(* IEC 61131-3 sources: repolevel_ST_code_completion/dataset/generation_context_ground_truth/Robotics_DynamicModel, 15 files *)

(* ---- SMC_Frame_ApplyWrench.st ---- *)
VAR
    mR_ : SM3M.SMC_Matrix3;
    wTmp0 : SM3M.SMC_VECTOR3D;
    wTmp1 : SM3M.SMC_VECTOR3D;
END_VAR

/// Applies a coordinate transformation T_ab to a wrench vector F_a in se(3).
///       |mR^T  mR^T*[vT]^T|
/// F_b = |                 | F_a
///       | 0         mR^T  |
FUNCTION SMC_Frame_ApplyWrench
VAR_IN_OUT
    /// Wrench vector in b frame coordinates.
	F_b : WrenchVec;
END_VAR
VAR_IN_OUT CONSTANT
    /// Orientation and position of the b frame
    /// in a frame coordinates.
	T_ab : SM3M.SMC_Frame;
    /// Wrench vector in a frame coordinates.
	F_a : WrenchVec;
END_VAR
VAR
    mR_ : SM3M.SMC_Matrix3;
    wTmp0 : SM3M.SMC_VECTOR3D;
    wTmp1 : SM3M.SMC_VECTOR3D;
END_VAR

(* ---- DynModel_Scara2_Z.st ---- *)
VAR CONSTANT
	/// Degrees of freedom.
	DOF : DINT := 3;
	/// All length values in [m]
	armOneLength : LREAL := 0.4;
	armTwoLength : LREAL := 0.3;
	baseHeight : LREAL := 0.6;
	armOneHeight : LREAL := 0.06;
	armTwoHeight : LREAL := 0.06;
	zAxisLength : LREAL := 0.3;
	zAxisOffset : LREAL := -0.05;
	/// All mass values in [kg]
	armOneMass : LREAL := 3;
	armTwoMass : LREAL := 4;
	zAxisMass : LREAL := 1;

	/// The home position of all link frames. |aM[i]| contains
    /// the frame of the ith link expressed in the coordinates of the
    /// (i-1)th link frame.
    /// All frames are expected to be situated at the link's center
    /// of mass.
    m_aM : ARRAY[0..SMRB.MAX_VEC_DIM] OF SM3M.SMC_Frame := [
        /// All values of vT in [m]
        ///
        /// The center of mass of arm 1 expressed in the base coordinate system 0:
        (mR:= (
            aElems:= [
                1, 0, 0,
                0, -1, 0,
                0, 0, -1]),
         vT:= (dX:= armOneLength / 2.0, dY:= 0, dZ:= baseHeight + armOneHeight / 2.0)),
        /// The center of mass of arm 2 expressed in the coordinate system of arm 1:
        (mR:= (
            aElems:= [
                1, 0, 0,
                0, 1, 0,
                0, 0, 1]),
         vT:= (dX:= armOneLength / 2.0 + armTwoLength / 2.0, dY:= 0, dZ:= armOneHeight / 2.0 + armTwoHeight / 2.0)),
        /// The center of mass of the z-axis expressed in the coordinate system of arm 2:
        (mR:= (
            aElems:= [
                1, 0, 0,
                0, 1, 0,
                0, 0, 1]),
         vT:= (dX:= armTwoLength / 2.0, dY:= 0, dZ:= zAxisLength / 2.0 - armTwoHeight / 2.0 + zAxisOffset)),
        /// One additional array entry, to handle an arbitrary load at the TCP, expressed
		/// in the coordinate system of the z-axis.
        (mR:= (
            aElems:= [
                1, 0, 0,
                0, 1, 0,
                0, 0, 1]),
         vT:= (dX:= 0, dY:= 0, dZ:= - zAxisLength / 2.0))];

	/// The spatial inertia matrices of all links, expressed in the
    /// respectives link's frame.
    m_aG : ARRAY[0..SMRB.MAX_VEC_DIM-1] OF SMDYN.DynSpatialInertia := [
        /// All inertia values in [kg m²]
        /// and all mass values in [kg]
        /// Arm 1
        (I:= (
            aElems:= [
                0, 0, 0,
                0, 1/12.0 * armOneMass * armOneLength * armOneLength, 0,
                0, 0, 1/12.0 * armOneMass * armOneLength * armOneLength]),
         m:= armOneMass),
        /// Arm 2
        (I:= (
            aElems:= [
                0, 0, 0,
                0, 1/12.0 * armTwoMass * armTwoLength * armTwoLength, 0,
                0, 0, 1/12.0 * armTwoMass * armTwoLength * armTwoLength]),
         m:= armTwoMass),
        /// z-axis
        (I:= (
            aElems:= [
                1/12.0 * zAxisMass * zAxisLength * zAxisLength, 0, 0,
                0, 1/12.0 * zAxisMass * zAxisLength * zAxisLength, 0,
                0, 0, 0]),
         m:= zAxisMass)];

	/// The screw axes of all joints, expressed in the base frame.
    m_aS : ARRAY[0..SMRB.MAX_VEC_DIM-1] OF TwistVec := [
		/// Angular velocities in [rad/s] and linear velocities in [m/s].
        /// Screw axis of arm 1
        (w:= (dX:= 0, dY:= 0, dZ:= 1),
         v:= (dX:= 0, dY:= 0, dZ:= 0)),
        /// Screw axis of arm 2
        (w:= (dX:= 0, dY:= 0, dZ:= 1),
         v:= (dX:= 0, dY:= -armOneLength, dZ:= 0)),
        /// Screw axis of the z-axis
        (w:= (dX:= 0, dY:= 0, dZ:= 0),
         v:= (dX:= 0, dY:= 0, dZ:= 1))];
END_VAR
VAR
    /// The home position of all link frames. |m_aM_inv[i]| contains
    /// the frame of the (i-1) link expressed in the coordinates of the
    /// ith link frame.
    /// All frames are expected to be situated at the link's center
    /// of mass.
    m_aM_inv : ARRAY[0..SM3M.SMC_MAX_VEC_DIM] OF SM3M.SMC_Frame;
    /// The screw axes of all joints, expressed in the link's frame.
    m_aA : ARRAY[0..SM3M.SMC_MAX_VEC_DIM-1] OF TwistVec;
END_VAR

(* ---- DynModel_Scara2_Z_AxesStateToTorque.st ---- *)
VAR
	m_aM_inv : ARRAY[0..SM3M.SMC_MAX_VEC_DIM] OF SM3M.SMC_Frame;
    /// The screw axes of all joints, expressed in the link's frame.
    m_aA : ARRAY[0..SM3M.SMC_MAX_VEC_DIM-1] OF TwistVec;
    convertedAxesState : SM3M.SMC_DynVecState;
	i : DINT;
END_VAR

VAR CONSTANT
/// Degrees of freedom.
	DOF : DINT := 3;
	/// All length values in [m]
	armOneLength : LREAL := 0.4;
	armTwoLength : LREAL := 0.3;
	baseHeight : LREAL := 0.6;
	armOneHeight : LREAL := 0.06;
	armTwoHeight : LREAL := 0.06;
	zAxisLength : LREAL := 0.3;
	zAxisOffset : LREAL := -0.05;
	/// All mass values in [kg]
	armOneMass : LREAL := 3;
	armTwoMass : LREAL := 4;
	zAxisMass : LREAL := 1;

	/// The home position of all link frames. |aM[i]| contains
    /// the frame of the ith link expressed in the coordinates of the
    /// (i-1)th link frame.
    /// All frames are expected to be situated at the link's center
    /// of mass.
    m_aM : ARRAY[0..SMRB.MAX_VEC_DIM] OF SM3M.SMC_Frame := [
        /// All values of vT in [m]
        ///
        /// The center of mass of arm 1 expressed in the base coordinate system 0:
        (mR:= (
            aElems:= [
                1, 0, 0,
                0, -1, 0,
                0, 0, -1]),
         vT:= (dX:= armOneLength / 2.0, dY:= 0, dZ:= baseHeight + armOneHeight / 2.0)),
        /// The center of mass of arm 2 expressed in the coordinate system of arm 1:
        (mR:= (
            aElems:= [
                1, 0, 0,
                0, 1, 0,
                0, 0, 1]),
         vT:= (dX:= armOneLength / 2.0 + armTwoLength / 2.0, dY:= 0, dZ:= armOneHeight / 2.0 + armTwoHeight / 2.0)),
        /// The center of mass of the z-axis expressed in the coordinate system of arm 2:
        (mR:= (
            aElems:= [
                1, 0, 0,
                0, 1, 0,
                0, 0, 1]),
         vT:= (dX:= armTwoLength / 2.0, dY:= 0, dZ:= zAxisLength / 2.0 - armTwoHeight / 2.0 + zAxisOffset)),
        /// One additional array entry, to handle an arbitrary load at the TCP, expressed
		/// in the coordinate system of the z-axis.
        (mR:= (
            aElems:= [
                1, 0, 0,
                0, 1, 0,
                0, 0, 1]),
         vT:= (dX:= 0, dY:= 0, dZ:= - zAxisLength / 2.0))];

	/// The spatial inertia matrices of all links, expressed in the
    /// respectives link's frame.
    m_aG : ARRAY[0..SMRB.MAX_VEC_DIM-1] OF SMDYN.DynSpatialInertia := [
        /// All inertia values in [kg m²]
        /// and all mass values in [kg]
        /// Arm 1
        (I:= (
            aElems:= [
                0, 0, 0,
                0, 1/12.0 * armOneMass * armOneLength * armOneLength, 0,
                0, 0, 1/12.0 * armOneMass * armOneLength * armOneLength]),
         m:= armOneMass),
        /// Arm 2
        (I:= (
            aElems:= [
                0, 0, 0,
                0, 1/12.0 * armTwoMass * armTwoLength * armTwoLength, 0,
                0, 0, 1/12.0 * armTwoMass * armTwoLength * armTwoLength]),
         m:= armTwoMass),
        /// z-axis
        (I:= (
            aElems:= [
                1/12.0 * zAxisMass * zAxisLength * zAxisLength, 0, 0,
                0, 1/12.0 * zAxisMass * zAxisLength * zAxisLength, 0,
                0, 0, 0]),
         m:= zAxisMass)];

	/// The screw axes of all joints, expressed in the base frame.
    m_aS : ARRAY[0..SMRB.MAX_VEC_DIM-1] OF TwistVec := [
		/// Angular velocities in [rad/s] and linear velocities in [m/s].
        /// Screw axis of arm 1
        (w:= (dX:= 0, dY:= 0, dZ:= 1),
         v:= (dX:= 0, dY:= 0, dZ:= 0)),
        /// Screw axis of arm 2
        (w:= (dX:= 0, dY:= 0, dZ:= 1),
         v:= (dX:= 0, dY:= -armOneLength, dZ:= 0)),
        /// Screw axis of the z-axis
        (w:= (dX:= 0, dY:= 0, dZ:= 0),
         v:= (dX:= 0, dY:= 0, dZ:= 1))];
END_VAR

ConvertAxesState(convertedAxesState, axesState);

SolveOpenChainDynamics(
	torque:= torque,
	uv:= convertedAxesState,
	g:= addParams.g,
	load:= addParams.load);

AxesStateToTorque := SMC_NO_ERROR;

(* ---- DynModel_Scara2_Z_ConvertAxesState.st ---- *)
VAR
    i : DINT;
	m_aM_inv : ARRAY[0..SM3M.SMC_MAX_VEC_DIM] OF SM3M.SMC_Frame;
    /// The screw axes of all joints, expressed in the link's frame.
    m_aA : ARRAY[0..SM3M.SMC_MAX_VEC_DIM-1] OF TwistVec;
END_VAR
VAR CONSTANT
/// Degrees of freedom.
	DOF : DINT := 3;
	/// All length values in [m]
	armOneLength : LREAL := 0.4;
	armTwoLength : LREAL := 0.3;
	baseHeight : LREAL := 0.6;
	armOneHeight : LREAL := 0.06;
	armTwoHeight : LREAL := 0.06;
	zAxisLength : LREAL := 0.3;
	zAxisOffset : LREAL := -0.05;
	/// All mass values in [kg]
	armOneMass : LREAL := 3;
	armTwoMass : LREAL := 4;
	zAxisMass : LREAL := 1;

	/// The home position of all link frames. |aM[i]| contains
    /// the frame of the ith link expressed in the coordinates of the
    /// (i-1)th link frame.
    /// All frames are expected to be situated at the link's center
    /// of mass.
    m_aM : ARRAY[0..SMRB.MAX_VEC_DIM] OF SM3M.SMC_Frame := [
        /// All values of vT in [m]
        ///
        /// The center of mass of arm 1 expressed in the base coordinate system 0:
        (mR:= (
            aElems:= [
                1, 0, 0,
                0, -1, 0,
                0, 0, -1]),
         vT:= (dX:= armOneLength / 2.0, dY:= 0, dZ:= baseHeight + armOneHeight / 2.0)),
        /// The center of mass of arm 2 expressed in the coordinate system of arm 1:
        (mR:= (
            aElems:= [
                1, 0, 0,
                0, 1, 0,
                0, 0, 1]),
         vT:= (dX:= armOneLength / 2.0 + armTwoLength / 2.0, dY:= 0, dZ:= armOneHeight / 2.0 + armTwoHeight / 2.0)),
        /// The center of mass of the z-axis expressed in the coordinate system of arm 2:
        (mR:= (
            aElems:= [
                1, 0, 0,
                0, 1, 0,
                0, 0, 1]),
         vT:= (dX:= armTwoLength / 2.0, dY:= 0, dZ:= zAxisLength / 2.0 - armTwoHeight / 2.0 + zAxisOffset)),
        /// One additional array entry, to handle an arbitrary load at the TCP, expressed
		/// in the coordinate system of the z-axis.
        (mR:= (
            aElems:= [
                1, 0, 0,
                0, 1, 0,
                0, 0, 1]),
         vT:= (dX:= 0, dY:= 0, dZ:= - zAxisLength / 2.0))];

	/// The spatial inertia matrices of all links, expressed in the
    /// respectives link's frame.
    m_aG : ARRAY[0..SMRB.MAX_VEC_DIM-1] OF SMDYN.DynSpatialInertia := [
        /// All inertia values in [kg m²]
        /// and all mass values in [kg]
        /// Arm 1
        (I:= (
            aElems:= [
                0, 0, 0,
                0, 1/12.0 * armOneMass * armOneLength * armOneLength, 0,
                0, 0, 1/12.0 * armOneMass * armOneLength * armOneLength]),
         m:= armOneMass),
        /// Arm 2
        (I:= (
            aElems:= [
                0, 0, 0,
                0, 1/12.0 * armTwoMass * armTwoLength * armTwoLength, 0,
                0, 0, 1/12.0 * armTwoMass * armTwoLength * armTwoLength]),
         m:= armTwoMass),
        /// z-axis
        (I:= (
            aElems:= [
                1/12.0 * zAxisMass * zAxisLength * zAxisLength, 0, 0,
                0, 1/12.0 * zAxisMass * zAxisLength * zAxisLength, 0,
                0, 0, 0]),
         m:= zAxisMass)];

	/// The screw axes of all joints, expressed in the base frame.
    m_aS : ARRAY[0..SMRB.MAX_VEC_DIM-1] OF TwistVec := [
		/// Angular velocities in [rad/s] and linear velocities in [m/s].
        /// Screw axis of arm 1
        (w:= (dX:= 0, dY:= 0, dZ:= 1),
         v:= (dX:= 0, dY:= 0, dZ:= 0)),
        /// Screw axis of arm 2
        (w:= (dX:= 0, dY:= 0, dZ:= 1),
         v:= (dX:= 0, dY:= -armOneLength, dZ:= 0)),
        /// Screw axis of the z-axis
        (w:= (dX:= 0, dY:= 0, dZ:= 0),
         v:= (dX:= 0, dY:= 0, dZ:= 1))];
END_VAR

FOR i := 0 TO 2 DO
	CASE i OF
		0, 1:
			convertedAxesState.v.a[i] := axesState.v.a[i] * SM3M.SMC_FACTOR_DEG_TO_RAD;
			convertedAxesState.v_s.a[i] := axesState.v_s.a[i] * SM3M.SMC_FACTOR_DEG_TO_RAD;
			convertedAxesState.v_ss.a[i] := axesState.v_ss.a[i] * SM3M.SMC_FACTOR_DEG_TO_RAD;

		2:
			convertedAxesState.v.a[i] := axesState.v.a[i];
			convertedAxesState.v_s.a[i] := axesState.v_s.a[i];
			convertedAxesState.v_ss.a[i] := axesState.v_ss.a[i];
	END_CASE
END_FOR

convertedAxesState.v.n :=
convertedAxesState.v_s.n :=
convertedAxesState.v_ss.n := 3;

(* ---- DynModel_Scara2_Z_Init.st ---- *)
VAR CONSTANT
/// Degrees of freedom.
	DOF : DINT := 3;
	/// All length values in [m]
	armOneLength : LREAL := 0.4;
	armTwoLength : LREAL := 0.3;
	baseHeight : LREAL := 0.6;
	armOneHeight : LREAL := 0.06;
	armTwoHeight : LREAL := 0.06;
	zAxisLength : LREAL := 0.3;
	zAxisOffset : LREAL := -0.05;
	/// All mass values in [kg]
	armOneMass : LREAL := 3;
	armTwoMass : LREAL := 4;
	zAxisMass : LREAL := 1;

	/// The home position of all link frames. |aM[i]| contains
    /// the frame of the ith link expressed in the coordinates of the
    /// (i-1)th link frame.
    /// All frames are expected to be situated at the link's center
    /// of mass.
    m_aM : ARRAY[0..SMRB.MAX_VEC_DIM] OF SM3M.SMC_Frame := [
        /// All values of vT in [m]
        ///
        /// The center of mass of arm 1 expressed in the base coordinate system 0:
        (mR:= (
            aElems:= [
                1, 0, 0,
                0, -1, 0,
                0, 0, -1]),
         vT:= (dX:= armOneLength / 2.0, dY:= 0, dZ:= baseHeight + armOneHeight / 2.0)),
        /// The center of mass of arm 2 expressed in the coordinate system of arm 1:
        (mR:= (
            aElems:= [
                1, 0, 0,
                0, 1, 0,
                0, 0, 1]),
         vT:= (dX:= armOneLength / 2.0 + armTwoLength / 2.0, dY:= 0, dZ:= armOneHeight / 2.0 + armTwoHeight / 2.0)),
        /// The center of mass of the z-axis expressed in the coordinate system of arm 2:
        (mR:= (
            aElems:= [
                1, 0, 0,
                0, 1, 0,
                0, 0, 1]),
         vT:= (dX:= armTwoLength / 2.0, dY:= 0, dZ:= zAxisLength / 2.0 - armTwoHeight / 2.0 + zAxisOffset)),
        /// One additional array entry, to handle an arbitrary load at the TCP, expressed
		/// in the coordinate system of the z-axis.
        (mR:= (
            aElems:= [
                1, 0, 0,
                0, 1, 0,
                0, 0, 1]),
         vT:= (dX:= 0, dY:= 0, dZ:= - zAxisLength / 2.0))];

	/// The spatial inertia matrices of all links, expressed in the
    /// respectives link's frame.
    m_aG : ARRAY[0..SMRB.MAX_VEC_DIM-1] OF SMDYN.DynSpatialInertia := [
        /// All inertia values in [kg m²]
        /// and all mass values in [kg]
        /// Arm 1
        (I:= (
            aElems:= [
                0, 0, 0,
                0, 1/12.0 * armOneMass * armOneLength * armOneLength, 0,
                0, 0, 1/12.0 * armOneMass * armOneLength * armOneLength]),
         m:= armOneMass),
        /// Arm 2
        (I:= (
            aElems:= [
                0, 0, 0,
                0, 1/12.0 * armTwoMass * armTwoLength * armTwoLength, 0,
                0, 0, 1/12.0 * armTwoMass * armTwoLength * armTwoLength]),
         m:= armTwoMass),
        /// z-axis
        (I:= (
            aElems:= [
                1/12.0 * zAxisMass * zAxisLength * zAxisLength, 0, 0,
                0, 1/12.0 * zAxisMass * zAxisLength * zAxisLength, 0,
                0, 0, 0]),
         m:= zAxisMass)];

	/// The screw axes of all joints, expressed in the base frame.
    m_aS : ARRAY[0..SMRB.MAX_VEC_DIM-1] OF TwistVec := [
		/// Angular velocities in [rad/s] and linear velocities in [m/s].
        /// Screw axis of arm 1
        (w:= (dX:= 0, dY:= 0, dZ:= 1),
         v:= (dX:= 0, dY:= 0, dZ:= 0)),
        /// Screw axis of arm 2
        (w:= (dX:= 0, dY:= 0, dZ:= 1),
         v:= (dX:= 0, dY:= -armOneLength, dZ:= 0)),
        /// Screw axis of the z-axis
        (w:= (dX:= 0, dY:= 0, dZ:= 0),
         v:= (dX:= 0, dY:= 0, dZ:= 1))];
END_VAR
VAR
    i : DINT;
    M_ib_ : SM3M.SMC_Frame;
    M_ib : SM3M.SMC_Frame; // base frame expressed in ith frame
    m_aM_inv : ARRAY[0..SM3M.SMC_MAX_VEC_DIM] OF SM3M.SMC_Frame;
    /// The screw axes of all joints, expressed in the link's frame.
    m_aA : ARRAY[0..SM3M.SMC_MAX_VEC_DIM-1] OF TwistVec;
END_VAR

/// Initialize constant parameters that are used by the open chain dynamics algorithm:
/// - Calculate the inverse frames of the center of mass positions m_aM_inv from the
/// given center of mass positions m_aM.
/// - Calculate the screw axes of all joints m_aA (expressed in the link´s frame)
/// from the given screw axes m_aS, which are expressed in the base frame.
M_ib := SM3M.SMC_Math_Global_Constants.SMC_FRAME_IDENTITY;
i := 0;
WHILE i < DOF DO
    SM3M.SMC_Frame_Inverse(m_aM_inv[i], m_aM[i]);

    SM3M.SMC_Frame_Mult(M_ib_, m_aM_inv[i], M_ib);
    M_ib := M_ib_;
    SMC_Frame_ApplyTwist(m_aA[i], M_ib, m_aS[i]);

    i := i + 1;
END_WHILE

SM3M.SMC_Frame_Inverse(m_aM_inv[DOF], m_aM[DOF]);

(* ---- DynModel_Scara2_Z_SolveOpenChainDynamics.st ---- *)
VAR
    T : ARRAY[0..SM3M.SMC_MAX_VEC_DIM] OF SM3M.SMC_Frame;
    V : ARRAY[0..SM3M.SMC_MAX_VEC_DIM] OF TwistVec;
    V_t : ARRAY[0..SM3M.SMC_MAX_VEC_DIM] OF TwistVec;
    F : ARRAY[0..SM3M.SMC_MAX_VEC_DIM] OF WrenchVec;

    T_uq : SM3M.SMC_Frame;
    V_uq_s : TwistVec;
    V_t_uq_ss : TwistVec;
    V_prev : TwistVec;
    V_t_prev : TwistVec;
    V_t_brack : TwistVec;
    F_prev : WrenchVec;
    F_V : WrenchVec;
    F_V_t : WrenchVec;
    F_brack : WrenchVec;
    i : DINT;

    T_load_inv_Flange : SM3M.SMC_Frame;
    T_load_inv : SM3M.SMC_Frame;
    V_load : TwistVec;
    V_t_load : TwistVec;
    F_load : WrenchVec;
    F_V_load : WrenchVec;
    F_V_t_load : WrenchVec;
    F_brack_load : WrenchVec;
    m_aM_inv : ARRAY[0..SM3M.SMC_MAX_VEC_DIM] OF SM3M.SMC_Frame;
    /// The screw axes of all joints, expressed in the link's frame.
    m_aA : ARRAY[0..SM3M.SMC_MAX_VEC_DIM-1] OF TwistVec;
END_VAR
VAR CONSTANT
/// Degrees of freedom.
	DOF : DINT := 3;
	/// All length values in [m]
	armOneLength : LREAL := 0.4;
	armTwoLength : LREAL := 0.3;
	baseHeight : LREAL := 0.6;
	armOneHeight : LREAL := 0.06;
	armTwoHeight : LREAL := 0.06;
	zAxisLength : LREAL := 0.3;
	zAxisOffset : LREAL := -0.05;
	/// All mass values in [kg]
	armOneMass : LREAL := 3;
	armTwoMass : LREAL := 4;
	zAxisMass : LREAL := 1;

	/// The home position of all link frames. |aM[i]| contains
    /// the frame of the ith link expressed in the coordinates of the
    /// (i-1)th link frame.
    /// All frames are expected to be situated at the link's center
    /// of mass.
    m_aM : ARRAY[0..SMRB.MAX_VEC_DIM] OF SM3M.SMC_Frame := [
        /// All values of vT in [m]
        ///
        /// The center of mass of arm 1 expressed in the base coordinate system 0:
        (mR:= (
            aElems:= [
                1, 0, 0,
                0, -1, 0,
                0, 0, -1]),
         vT:= (dX:= armOneLength / 2.0, dY:= 0, dZ:= baseHeight + armOneHeight / 2.0)),
        /// The center of mass of arm 2 expressed in the coordinate system of arm 1:
        (mR:= (
            aElems:= [
                1, 0, 0,
                0, 1, 0,
                0, 0, 1]),
         vT:= (dX:= armOneLength / 2.0 + armTwoLength / 2.0, dY:= 0, dZ:= armOneHeight / 2.0 + armTwoHeight / 2.0)),
        /// The center of mass of the z-axis expressed in the coordinate system of arm 2:
        (mR:= (
            aElems:= [
                1, 0, 0,
                0, 1, 0,
                0, 0, 1]),
         vT:= (dX:= armTwoLength / 2.0, dY:= 0, dZ:= zAxisLength / 2.0 - armTwoHeight / 2.0 + zAxisOffset)),
        /// One additional array entry, to handle an arbitrary load at the TCP, expressed
		/// in the coordinate system of the z-axis.
        (mR:= (
            aElems:= [
                1, 0, 0,
                0, 1, 0,
                0, 0, 1]),
         vT:= (dX:= 0, dY:= 0, dZ:= - zAxisLength / 2.0))];

	/// The spatial inertia matrices of all links, expressed in the
    /// respectives link's frame.
    m_aG : ARRAY[0..SMRB.MAX_VEC_DIM-1] OF SMDYN.DynSpatialInertia := [
        /// All inertia values in [kg m²]
        /// and all mass values in [kg]
        /// Arm 1
        (I:= (
            aElems:= [
                0, 0, 0,
                0, 1/12.0 * armOneMass * armOneLength * armOneLength, 0,
                0, 0, 1/12.0 * armOneMass * armOneLength * armOneLength]),
         m:= armOneMass),
        /// Arm 2
        (I:= (
            aElems:= [
                0, 0, 0,
                0, 1/12.0 * armTwoMass * armTwoLength * armTwoLength, 0,
                0, 0, 1/12.0 * armTwoMass * armTwoLength * armTwoLength]),
         m:= armTwoMass),
        /// z-axis
        (I:= (
            aElems:= [
                1/12.0 * zAxisMass * zAxisLength * zAxisLength, 0, 0,
                0, 1/12.0 * zAxisMass * zAxisLength * zAxisLength, 0,
                0, 0, 0]),
         m:= zAxisMass)];

	/// The screw axes of all joints, expressed in the base frame.
    m_aS : ARRAY[0..SMRB.MAX_VEC_DIM-1] OF TwistVec := [
		/// Angular velocities in [rad/s] and linear velocities in [m/s].
        /// Screw axis of arm 1
        (w:= (dX:= 0, dY:= 0, dZ:= 1),
         v:= (dX:= 0, dY:= 0, dZ:= 0)),
        /// Screw axis of arm 2
        (w:= (dX:= 0, dY:= 0, dZ:= 1),
         v:= (dX:= 0, dY:= -armOneLength, dZ:= 0)),
        /// Screw axis of the z-axis
        (w:= (dX:= 0, dY:= 0, dZ:= 0),
         v:= (dX:= 0, dY:= 0, dZ:= 1))];
END_VAR

SM3M.SMC_V3_Mult(V_t[0].v, g, -1);

T[DOF] := m_aM_inv[DOF];

i := 0;
WHILE i < DOF DO
    SMC_Frame_FromScrewAxisAngle(T_uq, m_aA[i], -uv.v.a[i]);
    SM3M.SMC_Frame_Mult(T[i], T_uq, m_aM_inv[i]);

    SMC_Frame_ApplyTwist(V_prev, T[i], V[i]);
    TwistVec_Scale(V_uq_s, m_aA[i], uv.v_s.a[i]);
    TwistVec_Add(V[i+1], V_prev, V_uq_s);

    SMC_Frame_ApplyTwist(V_t_prev, T[i], V_t[i]);
    Twist_Bracket_Twist(V_t_brack, V[i+1], m_aA[i]);
    TwistVec_Scale(V_t_brack, V_t_brack, uv.v_s.a[i]);
    TwistVec_Scale(V_t_uq_ss, m_aA[i], uv.v_ss.a[i]);
    TwistVec_Add(V_t[i+1], V_t_prev, V_t_brack);
    TwistVec_Add(V_t[i+1], V_t[i+1], V_t_uq_ss);

    i := i + 1;
END_WHILE

SM3M.SMC_Frame_Inverse(T_load_inv_Flange, load.CenterOfMassFrame);
SM3M.SMC_Frame_Mult(T_load_inv, T_load_inv_Flange, T[i]);

SMC_Frame_ApplyTwist(V_load, T_load_inv, V[i]);
SMC_Frame_ApplyTwist(V_t_load, T_load_inv, V_t[i]);
MatSI_ApplyTwist(F_V_t_load, load.Inertia, V_t_load);
MatSI_ApplyTwist(F_V_load, load.Inertia, V_load);
Twist_Bracket_Wrench(F_brack_load, V_load, F_V_load);

WrenchVec_Sub(F_load, F_V_t_load, F_brack_load);
SMC_Frame_ApplyWrench(F[DOF], T_load_inv_Flange, F_load);

WHILE i > 0 DO
    SMC_Frame_ApplyWrench(F_prev, T[i], F[i]);
    MatSI_ApplyTwist(F_V_t, m_aG[i-1], V_t[i]);
    MatSI_ApplyTwist(F_V, m_aG[i-1], V[i]);
    Twist_Bracket_Wrench(F_brack, V[i], F_V);

    WrenchVec_Add(F[i-1], F_prev, F_V_t);
    WrenchVec_Sub(F[i-1], F[i-1], F_brack);

    torque.a[i-1] := Wrench_Dot_Twist(F[i-1], m_aA[i-1]);

    i := i - 1;
END_WHILE

torque.n := DOF;

(* ---- SMC_Frame_ApplyTwist.st ---- *)
VAR
    vTmp : SM3M.SMC_VECTOR3D;
END_VAR

SM3M.SMC_Matrix3_Apply(V_a.w, T_ab.mR, V_b.w);
SM3M.SMC_Matrix3_Apply(V_a.v, T_ab.mR, V_b.v);
SM3M.SMC_V3_Cross(vTmp, T_ab.vT, V_a.w);
SM3M.SMC_V3_Add(V_a.v, V_a.v, vTmp);

(* ---- SMC_Frame_FromScrewAxisAngle.st ---- *)
VAR
    wv : SM3M.SMC_VECTOR3D;
    w2v : SM3M.SMC_VECTOR3D;
    wt : SM3M.SMC_VECTOR3D;
END_VAR

SM3M.SMC_V3_Cross(wv, A.w, A.v);
SM3M.SMC_V3_Cross(w2v, A.w, wv);

SM3M.SMC_V3_Mult(f.vT, A.v, theta);
SM3M.SMC_V3_MAdd(f.vT, f.vT, wv, (1 - COS(theta)));
SM3M.SMC_V3_MAdd(f.vT, f.vT, w2v, (theta - SIN(theta)));

SM3M.SMC_V3_Mult(wt, A.w, theta);
SM3M.SMC_Matrix3_FromAxisAngle(f.mR, wt);

(* ---- SMC_OpenChainKinematics_SolveForward.st ---- *)
VAR
    i : UDINT;
    fTmp : SM3M.SMC_Frame;
    afCur : ARRAY[0..1] OF SM3M.SMC_Frame;
END_VAR

i := TO_UDINT(vJoints.n);
afCur[i AND 1] := fTCP_init;
WHILE i > 0 DO
    SMC_Frame_FromScrewAxisAngle(fTmp, aS[i-1], vJoints.a[i-1]);
    SM3M.SMC_Frame_Mult(afCur[(i-1) AND 1], fTmp, afCur[i AND 1]);

    i := i - 1;
END_WHILE

fTCP := afCur[0];

(* ---- Test_DynModel_Scara2_Z.st ---- *)
VAR
	m_dynModel : DynModel_Scara2_Z;
END_VAR
VAR CONSTANT
	/// Frame of the initial robot position.
	ZERO_TCP_FRAME : SM3M.SMC_Frame := (
        mR:= (
            aElems:= [
                1, 0, 0,
                0, 1, 0,
                0, 0, 1]),
        vT:= (
			dX:= m_dynModel.armOneLength + m_dynModel.armTwoLength,
			dY:= 0,
			dZ:= - m_dynModel.baseHeight - m_dynModel.armOneHeight - m_dynModel.zAxisOffset));
END_VAR

(* ---- Test_DynModel_Scara2_Z_CheckScrewAxis.st ---- *)
VAR
	state : INT;
	done : BOOL;
	error : BOOL;

	axisPos : TRAFO.AXISPOS_REF;
END_VAR
VAR CONSTANT
	EPS : LREAL := 1E-10;
END_VAR

m_dynModel.Init();

WHILE NOT done AND NOT error DO
	CASE state OF
		0:
			axisPos.a0 := 0;	/// [°]
			axisPos.a1 := 0;	/// [°]
			axisPos.a2 := 0;	/// [m]

			IF IsScrewAxisAndKinematicEqual(axisPos, EPS) THEN
				state := state + 10;
			ELSE
				error := TRUE;
			END_IF

		10:
			axisPos.a0 := 0;	/// [°]
			axisPos.a1 := 90;	/// [°]
			axisPos.a2 := 0.03;	/// [m]

			IF IsScrewAxisAndKinematicEqual(axisPos, EPS) THEN
				state := state + 10;
			ELSE
				error := TRUE;
			END_IF

		20:
			axisPos.a0 := 45;	/// [°]
			axisPos.a1 := -50;	/// [°]
			axisPos.a2 := -0.01;/// [m]

			IF IsScrewAxisAndKinematicEqual(axisPos, EPS) THEN
				state := state + 10;
			ELSE
				error := TRUE;
			END_IF

		30:
			done := TRUE;
	END_CASE
END_WHILE

CheckScrewAxis := done AND NOT error;

(* ---- Test_DynModel_Scara2_Z_CheckStandstillTorque.st ---- *)
VAR
	expectedTorque : SM3M.SMC_Vec;
	calculatedTorque : SM3M.SMC_Vec;
	axesState : SM3M.SMC_DynVecState;
	addParams : SMDYN.DynamicsParams;
	i : DINT;
END_VAR
VAR CONSTANT
	EPSILON : LREAL := 1E-10;
END_VAR

m_dynModel.Init();

/// All axes in zero position.
axesState.v.a[0] := 0;
axesState.v.a[1] := 0;
axesState.v.a[2] := 0;
axesState.v.n := axesState.v_s.n := axesState.v_ss.n := 3;

/// Gravitational acceleration in [m/s²]
addParams.g.dZ := 9.81;

/// Expected torque of the revolute axis of arm 1 in [Nm]
expectedTorque.a[0] := 0;
/// Expected torque of the revolute axis of arm 2 in [Nm]
expectedTorque.a[1] := 0;
/// Expected force of the prismatic z-axis in [N]
expectedTorque.a[2] := - m_dynModel.zAxisMass * 9.81;
expectedTorque.n := 3;

m_dynModel.AxesStateToTorque(
	torque:= calculatedTorque,
	axesState:= axesState,
	addParams:= addParams);

CheckStandstillTorque := calculatedTorque.n = expectedTorque.n;
FOR i := 0 TO calculatedTorque.n - 1 DO
	CheckStandstillTorque := CheckStandstillTorque
							 AND_THEN ABS(calculatedTorque.a[i] - expectedTorque.a[i]) <= EPSILON;
END_FOR

(* ---- Test_DynModel_Scara2_Z_IsScrewAxisAndKinematicEqual.st ---- *)
VAR
	getKinematic : MC_ReadKinTransform;
	screwAxisResult : SM3M.SMC_Frame;
	convertedAxisPos : SM3M.SMC_Vec;
	kinematicResult : SM3M.SMC_Frame;
	cdNotUsed : TRAFO.CONFIGDATA;
END_VAR

convertedAxisPos.a[0] := axisPos.a0 * SM3M.SMC_FACTOR_DEG_TO_RAD;
convertedAxisPos.a[1] := axisPos.a1 * SM3M.SMC_FACTOR_DEG_TO_RAD;
convertedAxisPos.a[2] := axisPos.a2;
convertedAxisPos.n := 3;

SMC_OpenChainKinematics_SolveForward(
	fTCP:= screwAxisResult,
	aS:= m_dynModel.m_aS,
	vJoints:= convertedAxisPos,
	fTCP_init:= ZERO_TCP_FRAME);

getKinematic(
	AxisGroup:= AxisGroup,
	Enable:= TRUE);

IF getKinematic.Valid AND_THEN getKinematic.KinTransform <> 0 THEN
	getKinematic.KinTransform.AxesToCartesian(
		f:= kinematicResult,
		cd:= cdNotUsed,
		a:= axisPos);

	IsScrewAxisAndKinematicEqual :=
		ABS(screwAxisResult.vT.dX - kinematicResult.vT.dX) <= epsilon
		AND_THEN ABS(screwAxisResult.vT.dY- kinematicResult.vT.dY) <= epsilon
		AND_THEN ABS(screwAxisResult.vT.dZ - kinematicResult.vT.dZ) <= epsilon;
ELSE
	IsScrewAxisAndKinematicEqual := FALSE;
END_IF

(* ---- Twist_Bracket_Twist.st ---- *)
VAR
    v0 : SM3M.SMC_VECTOR3D;
    v1 : SM3M.SMC_VECTOR3D;
END_VAR

SM3M.SMC_V3_Cross(v0, V_lhs.v, V_rhs.w);
SM3M.SMC_V3_Cross(v1, V_lhs.w, V_rhs.v);
SM3M.SMC_V3_Cross(V_dst.w, V_lhs.w, V_rhs.w);
SM3M.SMC_V3_Add(V_dst.v, v0, v1);

(* ---- Twist_Bracket_Wrench.st ---- *)
VAR
    m0 : SM3M.SMC_VECTOR3D;
    m1 : SM3M.SMC_VECTOR3D;
END_VAR

SM3M.SMC_V3_Cross(m0, F_src.m, V_src.w);
SM3M.SMC_V3_Cross(m1, F_src.f, V_src.v);
SM3M.SMC_V3_Cross(F_dst.f, F_src.f, V_src.w);
SM3M.SMC_V3_Add(F_dst.m, m0, m1);
